{attribute addProperty BoxType "EL9210-0000-0016"}
{attribute addProperty Id "PowerOKAT %I*PowerOK_5B5BD03A810FuseErrorAT %I*FuseError_3E6D53D3810WcStateAT %I*WcState_98A4DF7520.250InfoDataAT %I*InfoData_192954DE1620"}
{attribute addProperty CRC "2885088535"}
{attribute addProperty SizeInBites "34"}
{attribute addProperty SizeInBytes "4.25"}
TYPE EL9210_B219644D :
STRUCT
	{attribute addProperty Name "PowerOK"}
	PowerOK : PowerOK_5B5BD03A;
	{attribute addProperty Name "FuseError"}
	FuseError : FuseError_3E6D53D3;
	{attribute addProperty Name "WcState"}
	WcState : WcState_98A4DF75;
	{attribute addProperty Name "InfoData"}
	InfoData : InfoData_192954DE;
END_STRUCT
END_TYPE

(* stored: Version 1.2.0.0, ProductVersion 3.1.4024.9
   DUT EL9210_B219644D: Id {f8b2d0a1-18ac-4ae5-aeb2-668db17f0106} *)
